// TIA Portal V17 export
// export: Created 2025-06-26T06:49:25.2887212Z, ExportSetting WithDefaults, DisplayName Totally Integrated Automation Portal, DisplayVersion V17 Update 8, DisplayName TIA Portal Openness, DisplayVersion V17 Update 8, DisplayName TIA Portal Version Control Interface, DisplayVersion V17, DisplayName STEP 7 Professional, DisplayVersion V17 Update 8, DisplayName STEP 7 Safety, DisplayVersion V17 Update 6, DisplayName WinCC Advanced, DisplayVersion V17 Update 8
DATA_BLOCK "DB_Misc"   // DB6
{ S7_Optimized_Access := 'TRUE' }
AUTHOR : Heaten
VERSION : 0.1
// stored: AutoNumber true, DBAccessibleFromOPCUA true, DBAccessibleFromWebserver true, IsOnlyStoredInLoadMemory false, IsRetainMemResEnabled false, IsWriteProtectedInAS false, MemoryReserve 100
   VAR
      EvaporatorDischargePressureMean : "stCalcSelect";   // Average of Evaporator A & B discharge pressures
      EvaporatorDischargeTemperatureMin { S7_SetPoint := 'True'} : "stCalcSelect";   // Smaller of Evaporator A & B discharge temperatures
      EvaporatorDischargeTemperatureMean { S7_SetPoint := 'True'} : "stCalcSelect";   // Average of Evaporator A & B discharge temperatures
      EvaporatorDischargePressureOffset : Real := 0.0;   // HBL-PT-04
   END_VAR
BEGIN
   EvaporatorDischargePressureMean.nMode := 5;
   EvaporatorDischargeTemperatureMin.nMode := 3;
   EvaporatorDischargeTemperatureMean.nMode := 5;
END_DATA_BLOCK
